// TIA Portal V19 export
FUNCTION_BLOCK "Gestion des sorties"   // FB3, LAD
BEGIN

REGION Network 1: Descente vérin élévation pièce
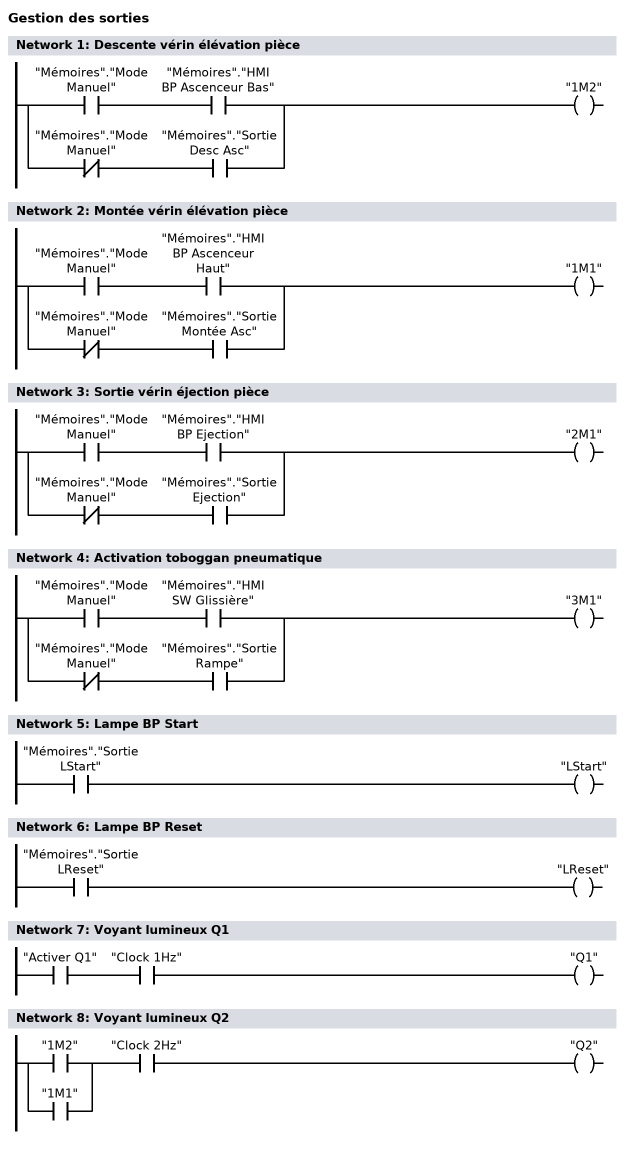
   RUNG wire#powerrail
      Contact( "Mémoires"."Mode Manuel" )
      Contact( "Mémoires"."HMI BP Ascenceur Bas" )
      wire#w1
      Coil( "1M2" )
   END_RUNG
   RUNG wire#powerrail
      I_Contact( "Mémoires"."Mode Manuel" )
      Contact( "Mémoires"."Sortie Desc Asc" )
   END_RUNG wire#w1
   // the same network as SCL:
   "1M2" := ("Mémoires"."Mode Manuel" AND "Mémoires"."HMI BP Ascenceur Bas") OR (NOT "Mémoires"."Mode Manuel" AND "Mémoires"."Sortie Desc Asc");
END_REGION

REGION Network 2: Montée vérin élévation pièce
   RUNG wire#powerrail
      Contact( "Mémoires"."Mode Manuel" )
      Contact( "Mémoires"."HMI BP Ascenceur Haut" )
      wire#w1
      Coil( "1M1" )
   END_RUNG
   RUNG wire#powerrail
      I_Contact( "Mémoires"."Mode Manuel" )
      Contact( "Mémoires"."Sortie Montée Asc" )
   END_RUNG wire#w1
   // the same network as SCL:
   "1M1" := ("Mémoires"."Mode Manuel" AND "Mémoires"."HMI BP Ascenceur Haut") OR (NOT "Mémoires"."Mode Manuel" AND "Mémoires"."Sortie Montée Asc");
END_REGION

REGION Network 3: Sortie vérin éjection pièce
   RUNG wire#powerrail
      Contact( "Mémoires"."Mode Manuel" )
      Contact( "Mémoires"."HMI BP Ejection" )
      wire#w1
      Coil( "2M1" )
   END_RUNG
   RUNG wire#powerrail
      I_Contact( "Mémoires"."Mode Manuel" )
      Contact( "Mémoires"."Sortie Ejection" )
   END_RUNG wire#w1
   // the same network as SCL:
   "2M1" := ("Mémoires"."Mode Manuel" AND "Mémoires"."HMI BP Ejection") OR (NOT "Mémoires"."Mode Manuel" AND "Mémoires"."Sortie Ejection");
END_REGION

REGION Network 4: Activation toboggan pneumatique
   RUNG wire#powerrail
      Contact( "Mémoires"."Mode Manuel" )
      Contact( "Mémoires"."HMI SW Glissière" )
      wire#w1
      Coil( "3M1" )
   END_RUNG
   RUNG wire#powerrail
      I_Contact( "Mémoires"."Mode Manuel" )
      Contact( "Mémoires"."Sortie Rampe" )
   END_RUNG wire#w1
   // the same network as SCL:
   "3M1" := ("Mémoires"."Mode Manuel" AND "Mémoires"."HMI SW Glissière") OR (NOT "Mémoires"."Mode Manuel" AND "Mémoires"."Sortie Rampe");
END_REGION

REGION Network 5: Lampe BP Start
   RUNG wire#powerrail
      Contact( "Mémoires"."Sortie LStart" )
      Coil( "LStart" )
   END_RUNG
   // the same network as SCL:
   "LStart" := "Mémoires"."Sortie LStart";
END_REGION

REGION Network 6: Lampe BP Reset
   RUNG wire#powerrail
      Contact( "Mémoires"."Sortie LReset" )
      Coil( "LReset" )
   END_RUNG
   // the same network as SCL:
   "LReset" := "Mémoires"."Sortie LReset";
END_REGION

REGION Network 7: Voyant lumineux Q1
   RUNG wire#powerrail
      Contact( "Activer Q1" )
      Contact( "Clock 1Hz" )
      Coil( "Q1" )
   END_RUNG
   // the same network as SCL:
   "Q1" := "Activer Q1" AND "Clock 1Hz";
END_REGION

REGION Network 8: Voyant lumineux Q2
   RUNG wire#powerrail
      Contact( "1M2" )
      wire#w1
      Contact( "Clock 2Hz" )
      Coil( "Q2" )
   END_RUNG
   RUNG wire#powerrail
      Contact( "1M1" )
   END_RUNG wire#w1
   // the same network as SCL:
   "Q2" := ("1M2" OR "1M1") AND "Clock 2Hz";
END_REGION
END_FUNCTION_BLOCK
